// TIA Portal project "Project1" (V16)

(* hardware
DEVICE "S7-1200 station_1"  S7-1200 Station
   slot 0: "Rack_0"  S7-1200 Rack  Rack  V1.0
   slot 1: "PLC_1"  CPU 1212C DC/DC/DC  6ES7 212-1AE31-0XB0  V3.0
   slot 2: "AI 4x13BIT_1"  SM 1231 AI4  6ES7 231-4HD30-0XB0  V1.0
   slot 3: "DI 8x24VDC_1"  SM 1221 DI8 x 24VDC  6ES7 221-1BF30-0XB0  V1.0
*)

// ===== PLC "PLC_1"  CPU 1212C DC/DC/DC =====

VAR_GLOBAL   // PLC tag table "Default tag table"
   "2 protection" AT %M10.6 : Bool;
   "3 protection" AT %M9.4 : Bool;
   "down" AT %M3.4 : Bool;
   "floor1" AT %Q1.1 : Bool;
   "floor2" AT %Q1.2 : Bool;
   "floor3" AT %Q1.3 : Bool;
   "floor4" AT %Q1.4 : Bool;
   "motor1" AT %Q0.1 : Bool;
   "motor2" AT %Q0.2 : Bool;
   "motor3" AT %Q0.3 : Bool;
   "motor4" AT %Q0.4 : Bool;
   "sensor1" AT %M4.1 : Bool;
   "sensor2" AT %M4.2 : Bool;
   "sensor3" AT %M4.3 : Bool;
   "sensor4" AT %M4.4 : Bool;
   "start1" AT %M0.1 : Bool;
   "start2" AT %M0.2 : Bool;
   "start3" AT %M0.3 : Bool;
   "start4" AT %M0.4 : Bool;
   "Tag_1" AT %M7.0 : Bool;
   "Tag_2" AT %M5.6 : Bool;
   "Tag_3" AT %M7.1 : Bool;
   "Tag_4" AT %M7.2 : Bool;
   "Tag_5" AT %M7.3 : Bool;
   "Tag_6" AT %M7.4 : Bool;
   "Tag_7" AT %M7.5 : Bool;
   "Tag_8" AT %M7.6 : Bool;
   "Tag_9" AT %M7.7 : Bool;
   "Tag_10" AT %M8.0 : Bool;
   "Tag_11" AT %M8.1 : Bool;
   "Tag_12" AT %M8.2 : Bool;
   "Tag_13" AT %M8.3 : Bool;
   "up" AT %M3.2 : Bool;
   "Tag_14" AT %M9.3 : Bool;
   "Tag_15" AT %M8.6 : Bool;
   "Tag_16" AT %M8.5 : Bool;
   "Tag_17" AT %M8.7 : Bool;
   "Tag_18" AT %M9.2 : Bool;
   "Tag_19" AT %M9.0 : Bool;
   "Tag_20" AT %M2.0 : Bool;
   "Tag_21" AT %M2.1 : Bool;
   "out1" AT %M1.1 : Bool;
   "out2" AT %M1.2 : Bool;
   "out3" AT %M1.3 : Bool;
   "out4" AT %M1.4 : Bool;
   "Tag_22" AT %M2.3 : Bool;
   "Tag_23" AT %M12.7 : Bool;
   "Tag_25" AT %M10.5 : Bool;
   "Tag_26" AT %M9.5 : Bool;
   "Tag_27" AT %M9.6 : Bool;
   "Tag_28" AT %M9.7 : Bool;
   "Tag_29" AT %M10.0 : Bool;
   "Tag_30" AT %M10.1 : Bool;
   "Tag_31" AT %M10.2 : Bool;
   "Tag_32" AT %M12.1 : Bool;
   "Tag_33" AT %M12.2 : Bool;
   "Tag_34" AT %M12.3 : Bool;
   "Tag_35" AT %M12.4 : Bool;
   "Tag_36" AT %M12.5 : Bool;
   "Tag_37" AT %M12.6 : Bool;
END_VAR

DATA_BLOCK "Data_START"   // DB1
{ S7_Optimized_Access := 'TRUE' }
VERSION : 0.1
// stored: InstanceOfName start
"start"
BEGIN
END_DATA_BLOCK

DATA_BLOCK "Data_up and down"   // DB2
{ S7_Optimized_Access := 'TRUE' }
VERSION : 0.1
// stored: InstanceOfName up and down
"up and down"
BEGIN
END_DATA_BLOCK

DATA_BLOCK "start_DB"   // DB3
{ S7_Optimized_Access := 'TRUE' }
VERSION : 0.1
// stored: InstanceOfName start
"start"
BEGIN
END_DATA_BLOCK

DATA_BLOCK "up and down_DB"   // DB4
{ S7_Optimized_Access := 'TRUE' }
VERSION : 0.1
// stored: InstanceOfName up and down
"up and down"
BEGIN
END_DATA_BLOCK

FUNCTION_BLOCK "up and down"   // FB1, LAD
TITLE = Up and Down
{ S7_Optimized_Access := 'TRUE' }
VERSION : 0.1
   VAR_TEMP   // added for the SCL form of the ladder/FBD networks
      _w1 : Bool;
      _w2 : Bool;
      _w3 : Bool;
      _w4 : Bool;
      _w5 : Bool;
   END_VAR
BEGIN

REGION Network 1: اولویت طبقه بالا
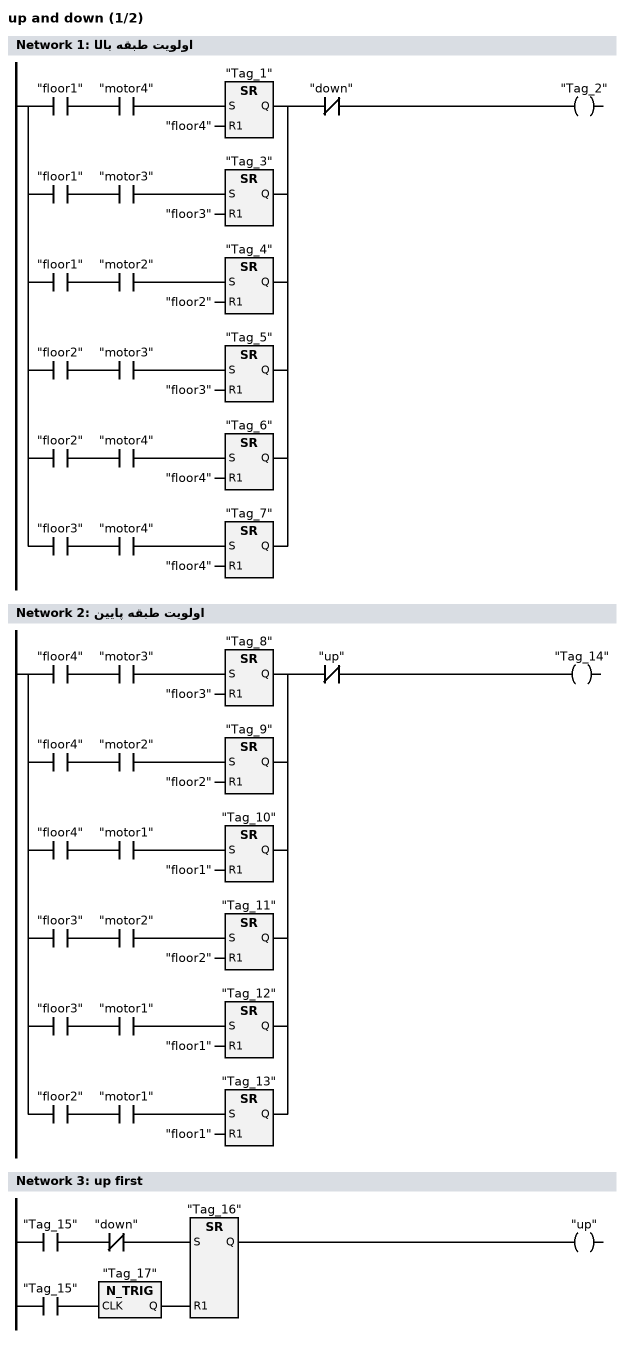
   RUNG wire#powerrail
      Contact( "floor1" )
      Contact( "motor4" )
      S_SR(operand := "Tag_1", r1 := "floor4")
      wire#w1
      I_Contact( "down" )
      Coil( "Tag_2" )
   END_RUNG
   RUNG wire#powerrail
      Contact( "floor1" )
      Contact( "motor3" )
      S_SR(operand := "Tag_3", r1 := "floor3")
   END_RUNG wire#w1
   RUNG wire#powerrail
      Contact( "floor1" )
      Contact( "motor2" )
      S_SR(operand := "Tag_4", r1 := "floor2")
   END_RUNG wire#w1
   RUNG wire#powerrail
      Contact( "floor2" )
      Contact( "motor3" )
      S_SR(operand := "Tag_5", r1 := "floor3")
   END_RUNG wire#w1
   RUNG wire#powerrail
      Contact( "floor2" )
      Contact( "motor4" )
      S_SR(operand := "Tag_6", r1 := "floor4")
   END_RUNG wire#w1
   RUNG wire#powerrail
      Contact( "floor3" )
      Contact( "motor4" )
      S_SR(operand := "Tag_7", r1 := "floor4")
   END_RUNG wire#w1
   // the same network as SCL:
   IF "floor1" AND "motor4" THEN
       "Tag_1" := TRUE;   // SR flip-flop
   END_IF;
   IF "floor4" THEN "Tag_1" := FALSE; END_IF;
   IF "floor1" AND "motor3" THEN
       "Tag_3" := TRUE;   // SR flip-flop
   END_IF;
   IF "floor3" THEN "Tag_3" := FALSE; END_IF;
   IF "floor1" AND "motor2" THEN
       "Tag_4" := TRUE;   // SR flip-flop
   END_IF;
   IF "floor2" THEN "Tag_4" := FALSE; END_IF;
   IF "floor2" AND "motor3" THEN
       "Tag_5" := TRUE;   // SR flip-flop
   END_IF;
   IF "floor3" THEN "Tag_5" := FALSE; END_IF;
   IF "floor2" AND "motor4" THEN
       "Tag_6" := TRUE;   // SR flip-flop
   END_IF;
   IF "floor4" THEN "Tag_6" := FALSE; END_IF;
   IF "floor3" AND "motor4" THEN
       "Tag_7" := TRUE;   // SR flip-flop
   END_IF;
   IF "floor4" THEN "Tag_7" := FALSE; END_IF;
   "Tag_2" := ("Tag_1" OR "Tag_3" OR "Tag_4" OR "Tag_5" OR "Tag_6" OR "Tag_7") AND NOT "down";
END_REGION

REGION Network 2: اولویت طبقه پایین
   RUNG wire#powerrail
      Contact( "floor4" )
      Contact( "motor3" )
      S_SR(operand := "Tag_8", r1 := "floor3")
      wire#w1
      I_Contact( "up" )
      Coil( "Tag_14" )
   END_RUNG
   RUNG wire#powerrail
      Contact( "floor4" )
      Contact( "motor2" )
      S_SR(operand := "Tag_9", r1 := "floor2")
   END_RUNG wire#w1
   RUNG wire#powerrail
      Contact( "floor4" )
      Contact( "motor1" )
      S_SR(operand := "Tag_10", r1 := "floor1")
   END_RUNG wire#w1
   RUNG wire#powerrail
      Contact( "floor3" )
      Contact( "motor2" )
      S_SR(operand := "Tag_11", r1 := "floor2")
   END_RUNG wire#w1
   RUNG wire#powerrail
      Contact( "floor3" )
      Contact( "motor1" )
      S_SR(operand := "Tag_12", r1 := "floor1")
   END_RUNG wire#w1
   RUNG wire#powerrail
      Contact( "floor2" )
      Contact( "motor1" )
      S_SR(operand := "Tag_13", r1 := "floor1")
   END_RUNG wire#w1
   // the same network as SCL:
   IF "floor4" AND "motor3" THEN
       "Tag_8" := TRUE;   // SR flip-flop
   END_IF;
   IF "floor3" THEN "Tag_8" := FALSE; END_IF;
   IF "floor4" AND "motor2" THEN
       "Tag_9" := TRUE;   // SR flip-flop
   END_IF;
   IF "floor2" THEN "Tag_9" := FALSE; END_IF;
   IF "floor4" AND "motor1" THEN
       "Tag_10" := TRUE;   // SR flip-flop
   END_IF;
   IF "floor1" THEN "Tag_10" := FALSE; END_IF;
   IF "floor3" AND "motor2" THEN
       "Tag_11" := TRUE;   // SR flip-flop
   END_IF;
   IF "floor2" THEN "Tag_11" := FALSE; END_IF;
   IF "floor3" AND "motor1" THEN
       "Tag_12" := TRUE;   // SR flip-flop
   END_IF;
   IF "floor1" THEN "Tag_12" := FALSE; END_IF;
   IF "floor2" AND "motor1" THEN
       "Tag_13" := TRUE;   // SR flip-flop
   END_IF;
   IF "floor1" THEN "Tag_13" := FALSE; END_IF;
   "Tag_14" := ("Tag_8" OR "Tag_9" OR "Tag_10" OR "Tag_11" OR "Tag_12" OR "Tag_13") AND NOT "up";
END_REGION

REGION Network 3: up first
   RUNG wire#powerrail
      Contact( "Tag_15" )
      I_Contact( "down" )
      S_SR(operand := "Tag_16", r1 := wire#w1)
      Coil( "up" )
   END_RUNG
   RUNG wire#powerrail
      Contact( "Tag_15" )
      N_Trig( "Tag_17" )
   END_RUNG wire#w1
   // the same network as SCL:
   #_w1 := NOT "Tag_15" AND "Tag_17";   // falling edge
   "Tag_17" := "Tag_15";
   IF "Tag_15" AND NOT "down" THEN
       "Tag_16" := TRUE;   // SR flip-flop
   END_IF;
   IF #_w1 THEN "Tag_16" := FALSE; END_IF;
   "up" := "Tag_16";
END_REGION

REGION Network 4: down first
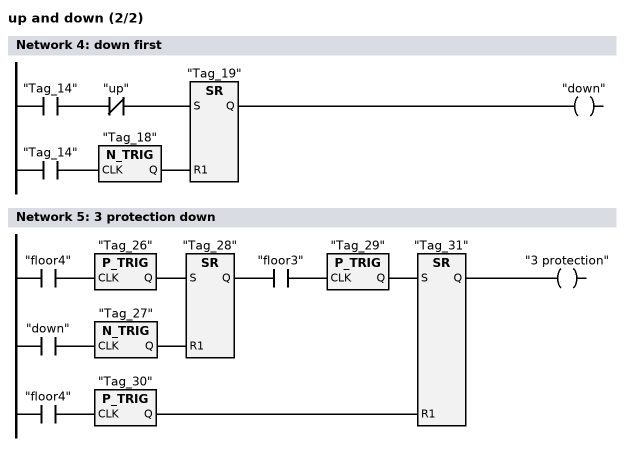
   RUNG wire#powerrail
      Contact( "Tag_14" )
      I_Contact( "up" )
      S_SR(operand := "Tag_19", r1 := wire#w1)
      Coil( "down" )
   END_RUNG
   RUNG wire#powerrail
      Contact( "Tag_14" )
      N_Trig( "Tag_18" )
   END_RUNG wire#w1
   // the same network as SCL:
   #_w1 := NOT "Tag_14" AND "Tag_18";   // falling edge
   "Tag_18" := "Tag_14";
   IF "Tag_14" AND NOT "up" THEN
       "Tag_19" := TRUE;   // SR flip-flop
   END_IF;
   IF #_w1 THEN "Tag_19" := FALSE; END_IF;
   "down" := "Tag_19";
END_REGION

REGION Network 5: 3 protection down
   RUNG wire#powerrail
      Contact( "floor4" )
      P_Trig( "Tag_26" )
      S_SR(operand := "Tag_28", r1 := wire#w1)
      Contact( "floor3" )
      P_Trig( "Tag_29" )
      S_SR(operand := "Tag_31", r1 := wire#w2)
      Coil( "3 protection" )
   END_RUNG
   RUNG wire#powerrail
      Contact( "down" )
      N_Trig( "Tag_27" )
   END_RUNG wire#w1
   RUNG wire#powerrail
      Contact( "floor4" )
      P_Trig( "Tag_30" )
   END_RUNG wire#w2
   // the same network as SCL:
   #_w1 := "floor4" AND NOT "Tag_26";   // rising edge
   "Tag_26" := "floor4";
   #_w2 := NOT "down" AND "Tag_27";   // falling edge
   "Tag_27" := "down";
   IF #_w1 THEN
       "Tag_28" := TRUE;   // SR flip-flop
   END_IF;
   IF #_w2 THEN "Tag_28" := FALSE; END_IF;
   #_w3 := "Tag_28" AND "floor3";
   #_w4 := #_w3 AND NOT "Tag_29";   // rising edge
   "Tag_29" := #_w3;
   #_w5 := "floor4" AND NOT "Tag_30";   // rising edge
   "Tag_30" := "floor4";
   IF #_w4 THEN
       "Tag_31" := TRUE;   // SR flip-flop
   END_IF;
   IF #_w5 THEN "Tag_31" := FALSE; END_IF;
   "3 protection" := "Tag_31";
END_REGION
END_FUNCTION_BLOCK

FUNCTION_BLOCK "start"   // FB2, LAD
{ S7_Optimized_Access := 'TRUE' }
VERSION : 0.1
   VAR_TEMP   // added for the SCL form of the ladder/FBD networks
      _w1 : Bool;
      _w2 : Bool;
      _w3 : Bool;
      _w4 : Bool;
      _w5 : Bool;
   END_VAR
BEGIN

REGION Network 1: 1
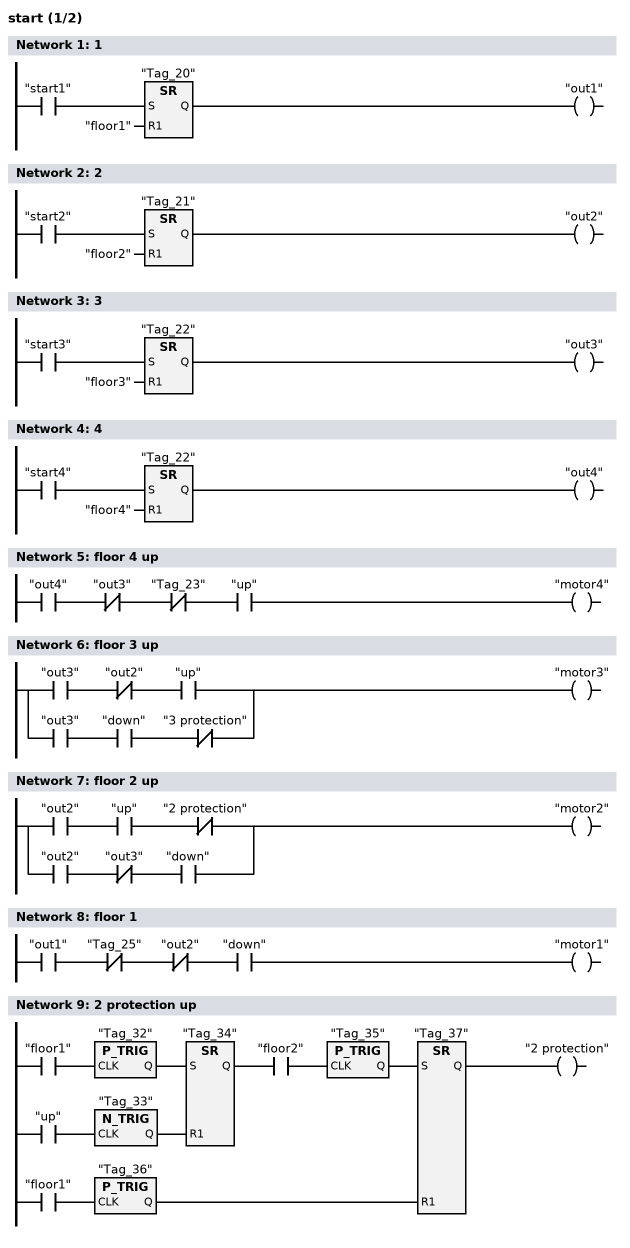
   RUNG wire#powerrail
      Contact( "start1" )
      S_SR(operand := "Tag_20", r1 := "floor1")
      Coil( "out1" )
   END_RUNG
   // the same network as SCL:
   IF "start1" THEN
       "Tag_20" := TRUE;   // SR flip-flop
   END_IF;
   IF "floor1" THEN "Tag_20" := FALSE; END_IF;
   "out1" := "Tag_20";
END_REGION

REGION Network 2: 2
   RUNG wire#powerrail
      Contact( "start2" )
      S_SR(operand := "Tag_21", r1 := "floor2")
      Coil( "out2" )
   END_RUNG
   // the same network as SCL:
   IF "start2" THEN
       "Tag_21" := TRUE;   // SR flip-flop
   END_IF;
   IF "floor2" THEN "Tag_21" := FALSE; END_IF;
   "out2" := "Tag_21";
END_REGION

REGION Network 3: 3
   RUNG wire#powerrail
      Contact( "start3" )
      S_SR(operand := "Tag_22", r1 := "floor3")
      Coil( "out3" )
   END_RUNG
   // the same network as SCL:
   IF "start3" THEN
       "Tag_22" := TRUE;   // SR flip-flop
   END_IF;
   IF "floor3" THEN "Tag_22" := FALSE; END_IF;
   "out3" := "Tag_22";
END_REGION

REGION Network 4: 4
   RUNG wire#powerrail
      Contact( "start4" )
      S_SR(operand := "Tag_22", r1 := "floor4")
      Coil( "out4" )
   END_RUNG
   // the same network as SCL:
   IF "start4" THEN
       "Tag_22" := TRUE;   // SR flip-flop
   END_IF;
   IF "floor4" THEN "Tag_22" := FALSE; END_IF;
   "out4" := "Tag_22";
END_REGION

REGION Network 5: floor 4 up
   RUNG wire#powerrail
      Contact( "out4" )
      I_Contact( "out3" )
      I_Contact( "Tag_23" )
      Contact( "up" )
      Coil( "motor4" )
   END_RUNG
   // the same network as SCL:
   "motor4" := "out4" AND NOT "out3" AND NOT "Tag_23" AND "up";
END_REGION

REGION Network 6: floor 3 up
   RUNG wire#powerrail
      Contact( "out3" )
      I_Contact( "out2" )
      Contact( "up" )
      wire#w1
      Coil( "motor3" )
   END_RUNG
   RUNG wire#powerrail
      Contact( "out3" )
      Contact( "down" )
      I_Contact( "3 protection" )
   END_RUNG wire#w1
   // the same network as SCL:
   "motor3" := ("out3" AND NOT "out2" AND "up") OR ("out3" AND "down" AND NOT "3 protection");
END_REGION

REGION Network 7: floor 2 up
   RUNG wire#powerrail
      Contact( "out2" )
      Contact( "up" )
      I_Contact( "2 protection" )
      wire#w1
      Coil( "motor2" )
   END_RUNG
   RUNG wire#powerrail
      Contact( "out2" )
      I_Contact( "out3" )
      Contact( "down" )
   END_RUNG wire#w1
   // the same network as SCL:
   "motor2" := ("out2" AND "up" AND NOT "2 protection") OR ("out2" AND NOT "out3" AND "down");
END_REGION

REGION Network 8: floor 1
   RUNG wire#powerrail
      Contact( "out1" )
      I_Contact( "Tag_25" )
      I_Contact( "out2" )
      Contact( "down" )
      Coil( "motor1" )
   END_RUNG
   // the same network as SCL:
   "motor1" := "out1" AND NOT "Tag_25" AND NOT "out2" AND "down";
END_REGION

REGION Network 9: 2 protection up
   RUNG wire#powerrail
      Contact( "floor1" )
      P_Trig( "Tag_32" )
      S_SR(operand := "Tag_34", r1 := wire#w1)
      Contact( "floor2" )
      P_Trig( "Tag_35" )
      S_SR(operand := "Tag_37", r1 := wire#w2)
      Coil( "2 protection" )
   END_RUNG
   RUNG wire#powerrail
      Contact( "up" )
      N_Trig( "Tag_33" )
   END_RUNG wire#w1
   RUNG wire#powerrail
      Contact( "floor1" )
      P_Trig( "Tag_36" )
   END_RUNG wire#w2
   // the same network as SCL:
   #_w1 := "floor1" AND NOT "Tag_32";   // rising edge
   "Tag_32" := "floor1";
   #_w2 := NOT "up" AND "Tag_33";   // falling edge
   "Tag_33" := "up";
   IF #_w1 THEN
       "Tag_34" := TRUE;   // SR flip-flop
   END_IF;
   IF #_w2 THEN "Tag_34" := FALSE; END_IF;
   #_w3 := "Tag_34" AND "floor2";
   #_w4 := #_w3 AND NOT "Tag_35";   // rising edge
   "Tag_35" := #_w3;
   #_w5 := "floor1" AND NOT "Tag_36";   // rising edge
   "Tag_36" := "floor1";
   IF #_w4 THEN
       "Tag_37" := TRUE;   // SR flip-flop
   END_IF;
   IF #_w5 THEN "Tag_37" := FALSE; END_IF;
   "2 protection" := "Tag_37";
END_REGION

REGION Network 10: 3 protection
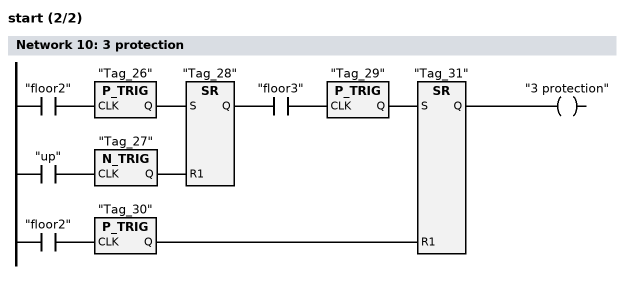
   RUNG wire#powerrail
      Contact( "floor2" )
      P_Trig( "Tag_26" )
      S_SR(operand := "Tag_28", r1 := wire#w1)
      Contact( "floor3" )
      P_Trig( "Tag_29" )
      S_SR(operand := "Tag_31", r1 := wire#w2)
      Coil( "3 protection" )
   END_RUNG
   RUNG wire#powerrail
      Contact( "up" )
      N_Trig( "Tag_27" )
   END_RUNG wire#w1
   RUNG wire#powerrail
      Contact( "floor2" )
      P_Trig( "Tag_30" )
   END_RUNG wire#w2
   // the same network as SCL:
   #_w1 := "floor2" AND NOT "Tag_26";   // rising edge
   "Tag_26" := "floor2";
   #_w2 := NOT "up" AND "Tag_27";   // falling edge
   "Tag_27" := "up";
   IF #_w1 THEN
       "Tag_28" := TRUE;   // SR flip-flop
   END_IF;
   IF #_w2 THEN "Tag_28" := FALSE; END_IF;
   #_w3 := "Tag_28" AND "floor3";
   #_w4 := #_w3 AND NOT "Tag_29";   // rising edge
   "Tag_29" := #_w3;
   #_w5 := "floor2" AND NOT "Tag_30";   // rising edge
   "Tag_30" := "floor2";
   IF #_w4 THEN
       "Tag_31" := TRUE;   // SR flip-flop
   END_IF;
   IF #_w5 THEN "Tag_31" := FALSE; END_IF;
   "3 protection" := "Tag_31";
END_REGION
END_FUNCTION_BLOCK

ORGANIZATION_BLOCK "Main"   // OB1, LAD, ProgramCycle
TITLE = "Main Program Sweep (Cycle)"
{ S7_Optimized_Access := 'TRUE' }
VERSION : 0.1
BEGIN

REGION Network 1
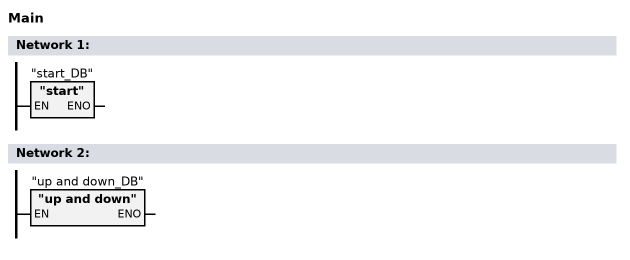
   RUNG wire#powerrail
      "start_DB"()
   END_RUNG
   // the same network as SCL:
   "start_DB"();   // "start"
END_REGION

REGION Network 2
   RUNG wire#powerrail
      "up and down_DB"()
   END_RUNG
   // the same network as SCL:
   "up and down_DB"();   // "up and down"
END_REGION
END_ORGANIZATION_BLOCK